PROGRAM main
  VAR
    HS101_Fill AT %IX0.0 : BOOL;
    HS102_Drain AT %IX0.1 : BOOL;
    LSH101_High AT %IX0.2 : BOOL;
    LSL102_Low AT %IX0.3 : BOOL;
    XV101_Fill AT %QX0.0 : BOOL;
    XV102_Drain AT %QX0.1 : BOOL;
  END_VAR

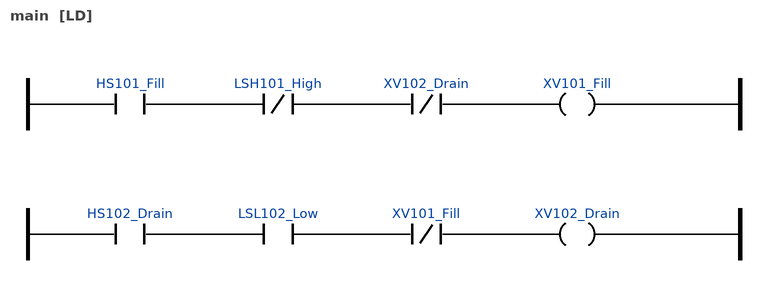
(* LD diagram, written out as Structured Text *)
XV101_Fill := HS101_Fill AND NOT LSH101_High AND NOT XV102_Drain;
XV102_Drain := HS102_Drain AND LSL102_Low AND NOT XV101_Fill;
END_PROGRAM
